FUNCTION_BLOCK FB_setupSlaveGravity
VAR_INPUT
END_VAR
VAR_OUTPUT
	o_Gravity:ARRAY[1..4,1..3] OF LREAL;
END_VAR
VAR
	m_armIdx :INT ;

	// current arm parameters
	m_armParams :ARRAY[1..5] OF LREAL;

END_VAR

METHOD getRegMat : BOOL
VAR_INPUT
	// joint position of setup joint, joint6-8
	setupAng :LREAL;
	q1: LREAL;
	q2: LREAL;
	q3: LREAL;
END_VAR

VAR
	gx, gy :LREAL;
	s0,c0,s1,c1,s2, c2,d3 :LREAL;
END_VAR

VAR_OUTPUT
	o_regMat:ARRAY[1..4,1..7] OF LREAL;
END_VAR
s0:= SIN(setUpAng);
c0:= COS(setUpAng);
s1:=SIN(q1);
c1:=COS(q1);
s2:=SIN(q2);
c2:=COS(q2);
d3:=q3;

// setup joint
o_regMat[1,1] :=c0;
o_regMat[1,2] :=-(c2*s0*d3+c0*c1*s2*d3);
o_regMat[1,3] :=  -c0*c1;
o_regMat[1,4] := -s0;
o_regMat[1,5] :=  -c0*s1;
o_regMat[1,6] := - (c0*c1*s2+c2*s0);
o_regMat[1,7] := s0*s2- c0*c1*c2 ;


// joint1
o_regMat[2,1] :=0;
o_regMat[2,2] :=s0*s1*s2*d3;
o_regMat[2,3] := s0*s1;
o_regMat[2,4] := 0;
o_regMat[2,5] := -s0*c1;
o_regMat[2,6] := s0*s1*s2;
o_regMat[2,7] := s0*c2*s1;

// joint2 
o_regMat[3,1] := 0;
o_regMat[3,2] := - (9.8*c0*s2*d3+9.8*s0*c1*c2*d3);
o_regMat[3,3] :=  0;
o_regMat[3,4] := 0;
o_regMat[3,5] :=  0;
o_regMat[3,6] := - (c0*s2+s0*c1*c2);
o_regMat[3,7] := s0*c1*s2- c0*c2  ;

// joint3
o_regMat[4,1] :=0;
o_regMat[4,2] := c0*c2 - s0*c1*s2;
o_regMat[4,3] :=  0;
o_regMat[4,4] := 0;
o_regMat[4,5] :=  0;
o_regMat[4,6] := 0;
o_regMat[4,7] := 0;
END_METHOD

METHOD init : BOOL
VAR_INPUT
	i_armIdx :INT;
END_VAR
m_armIdx :=i_armIdx;
END_METHOD

METHOD run : BOOL
VAR_IN_OUT CONSTANT
	// setup joint angle
	i_setupJntPos :Vec5d;
	
	// slave joint angle
	i_slaveJntPos :Vec8d;
	
	// instrument
	i_instruStatus :ST_InstruStatus;
END_VAR
VAR_OUTPUT
	// setup joint3 gravity
	o_setupJ3Gravity :LREAL;
	
	// setup joint5 gravity
	o_setupJ5Gravity :LREAL;
	
	// slave joint1-3 gravity
	o_slaveGravity : Vec3d;
END_VAR
VAR
	setupPos, q1, q2, q3 :LREAL;
	i,j:INT;
	
	gravityTrq :Vec4d;
	// gravity regression matrix
	regMat:ARRAY[1..4,1..7] OF LREAL;
END_VAR
setupPos:=i_setupJntPos[5];
q1 := i_slaveJntPos[1];
q2 := i_slaveJntPos[2];
q3 := i_slaveJntPos[3];


// get regression matrx
getRegMat(setupPos, q1, q2, q3, o_regMat=>regMat);

// determine current arm parameters
IF FALSE = i_instruStatus.m_ready THEN
	// arm only
	FOR i:=1 TO 7 DO
		m_armParams[i]:=GVLs_SetupSlaveArmDynamics.g_gravityParam[m_armIdx,i];
	END_FOR

// endoscope
ELSIF InstruType_endoscope = i_instruStatus.m_type THEN 
	FOR i:=1 TO 7 DO
		m_armParams[i]:=GVLs_SetupSlaveArmDynamics.g_gravityParam[m_armIdx,i]+GVLs_SetupSlaveArmDynamics.g_gravityEndoscope[i];
	END_FOR

// instrument
ELSE
	FOR i:=1 TO 7 DO
		m_armParams[i]:=GVLs_SetupSlaveArmDynamics.g_gravityParam[m_armIdx,i]+GVLs_SetupSlaveArmDynamics.g_gravityInstrument[i];
	END_FOR
// TODO:Trocar
END_IF

// calculate gravity torque
FOR i:=1 TO 4 DO
	gravityTrq[i]:=0;
	FOR j:=1 TO 7 DO
		gravityTrq[i]:=gravityTrq[i]+regMat[i,j]*m_armParams[j];
	END_FOR
END_FOR

o_setupJ5Gravity:=gravityTrq[1];
o_slaveGravity[1]:=gravityTrq[2];
o_slaveGravity[2]:=gravityTrq[3];
o_slaveGravity[3]:=gravityTrq[4];

// setup joint3 gravity fitting
o_setupJ3Gravity := setupJnt3Gravity(i_setupJntPos[3]);
END_METHOD

METHOD setupJnt3Gravity : LREAL
VAR_INPUT
	i_jnt3Pos :LREAL;
END_VAR
//TDDO calculate gravity of setup joint3 by polynomial fitting
END_METHOD

END_FUNCTION_BLOCK

(* stored: Version 1.1.0.1, ProductVersion 3.1.4024.12
   POU FB_setupSlaveGravity: Id {5452bfb6-8061-49fa-846a-f3728f3e7824}, SpecialFunc None
   Method getRegMat: Id {7045fe73-d3f1-4303-94f0-43372abb4236}
   Method init: Id {50ab6c0f-ea77-4dcf-ba79-983ca62b783b}
   Method run: Id {6d0c1aa2-0848-447c-a248-94105516dfb5}
   Method setupJnt3Gravity: Id {14b87259-982c-438c-9682-4b69bb2110c7} *)
